FUNCTION_BLOCK FB_OPCUA_Client_ReadVar EXTENDS FB_OPCUA_Client_Basic
VAR_INPUT
	iTargetSize	: UDINT;	// Size of local target variable
	pTarget		: pVoid;	// Address of local target variable
END_VAR
VAR_OUTPUT
END_VAR
VAR
	(* Declarations for UA_Read *)
	fbUA_Read				: UA_Read;
	stIndexRange			: ARRAY [1..nMaxIndexRange] OF ST_UAIndexRange;
	nIndexRangeCount		: UINT;
	stNodeAddInfo			: ST_UANodeAdditionalInfo;
	cbDataRead				: UDINT;
END_VAR
VAR PERSISTENT
END_VAR

CASE eState OF
	E_OPCUA_Client_Seq.Idle:
		IF (bExecute) THEN
			M_Init();
			eState := E_OPCUA_Client_Seq.CheckData;
		END_IF

	E_OPCUA_Client_Seq.CheckData:
		IF ((pTarget <> 0) AND (iTargetSize > 1)) THEN
			eState := E_OPCUA_Client_Seq.OpenSession;
		ELSE
			bError := TRUE;
			bBusy := FALSE;
			eState := E_OPCUA_Client_Seq.Done;
		END_IF

	E_OPCUA_Client_Seq.OpenSession:
		CASE M_OpenSession() OF
			E_Method.Done:	// Done
				eState := E_OPCUA_Client_Seq.GetNameSpace;
			E_Method.Error:	// Error
				eState := E_OPCUA_Client_Seq.Idle;			
		END_CASE

	E_OPCUA_Client_Seq.GetNameSpace:
		CASE M_GetNameSpace() OF
			E_Method.Done:	// Done
				eState := E_OPCUA_Client_Seq.GetNode;
			E_Method.Error:	// Error
				eState := E_OPCUA_Client_Seq.CloseSession;			
		END_CASE


	E_OPCUA_Client_Seq.GetNode:
		CASE M_GetNode() OF
			E_Method.Done:	// Done
				eState := E_OPCUA_Client_Seq.Read;
			E_Method.Error:	// Error
				eState := E_OPCUA_Client_Seq.CloseSession;			
		END_CASE


	E_OPCUA_Client_Seq.Read:
		CASE M_ReadVar() OF
			E_Method.Done:	// Done
				eState := E_OPCUA_Client_Seq.ReleaseNode;
			E_Method.Error:	// Error
				eState := E_OPCUA_Client_Seq.ReleaseNode;
		END_CASE

	E_OPCUA_Client_Seq.ReleaseNode:
		CASE M_ReleaseNode() OF
			E_Method.Done:	// Done
				eState := E_OPCUA_Client_Seq.CloseSession;
			E_Method.Error:	// Error
				eState := E_OPCUA_Client_Seq.CloseSession;
		END_CASE

	E_OPCUA_Client_Seq.CloseSession:
		CASE M_CloseSession() OF
			E_Method.Done:	// Done
				eState := E_OPCUA_Client_Seq.Done;
			E_Method.Error:	// Error
				eState := E_OPCUA_Client_Seq.Done;
		END_CASE
		
	E_OPCUA_Client_Seq.Done:
		bBusy := FALSE;
		IF (NOT bExecute) THEN
			bDone := FALSE;
			bError := FALSE;
			eState := E_OPCUA_Client_Seq.Idle;
		END_IF

	ELSE
		eState := E_OPCUA_Client_Seq.Idle;

END_CASE

METHOD PROTECTED M_Init : E_Method
VAR_INPUT
END_VAR
	
	SUPER^.M_Init();	

	stNodeAddInfo.nIndexRangeCount := nIndexRangeCount;
	stNodeAddInfo.stIndexRange := stIndexRange;

	M_Init := E_Method.Done;
END_METHOD

METHOD PROTECTED M_ReadVar : E_Method
VAR_INPUT
END_VAR

	fbUA_Read(	Execute := TRUE,
				ConnectionHdl := nConnectionHdl,
				NodeHdl := nNodeHdl,
				cbData := iTargetSize,
				stNodeAddInfo := stNodeAddInfo,
				pVariable := pTarget	);

	IF (fbUA_Read.Busy) THEN
		// Reading
		M_ReadVar := E_Method.Busy;
	ELSIF (fbUA_Read.Error) THEN
		// Error reading
		fbUA_Read(Execute := FALSE);
		bError := TRUE;
		nErrorID := fbUA_Read.ErrorID;
		M_ReadVar := E_Method.Error;
	ELSIF (fbUA_Read.Done) THEN
		// Data read OK
		fbUA_Read(Execute := FALSE);
		M_ReadVar := E_Method.Done;
	ELSE
		M_ReadVar := E_Method.Idle;			
	END_IF
END_METHOD

END_FUNCTION_BLOCK

(* stored: Version 1.1.0.1, ProductVersion 3.1.4024.2
   POU FB_OPCUA_Client_ReadVar: Id {61e9c7b1-4ad1-4da3-aac9-977f29b80f54}, SpecialFunc None
   Method M_Init: Id {e9e2e531-338f-4bad-9247-ca3b2d37fcf6}
   Method M_ReadVar: Id {1c72bd70-e86e-4320-9de5-f15492fabc7f} *)
